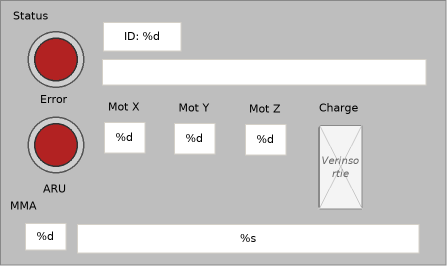
VISUALIZATION Visu2_Status  // 447x266
    Rectangle (-2,-2 447x266)
    Image (318,126 43x83), invisible if: fbAct1.xInInPos=0, image: Verinrentree
    Rectangle (320,150 37x38), "Going out", invisible if: fbAct1.xGoingOutNow=0
    Lamp1 (22,112 68x66), variable: fbBtn.xAru=0, style: Lamp-Lamp1-Red
    Lamp1 (23,25 66x69), variable: stParam.stStatus.xErreur, style: Lamp-Lamp1-Red
    Textfield (102,59 324x26), text variable: stParam.stStatus.sMessage, text list: 'ErrorList', text index: stParam.stStatus.iId
    Textfield (103,22 78x29), "ID: %d", text variable: stParam.stStatus.iId
    Label (299,93 80x30), "Charge"
    Image (319,125 43x84), invisible if: fbAct1.xInOutPos=0, image: Verinsortie
    Textfield (245,124 41x31), "%d", text variable: fbMotorZ.fbAxisRef.NcToPlc.ActPos
    Label (225,94 80x30), "Mot Z"
    Label (154,93 80x30), "Mot Y"
    Textfield (174,123 41x31), "%d", text variable: fbMotorY.fbAxisRef.NcToPlc.ActPos
    Label (84,92 80x30), "Mot X"
    Textfield (104,122 41x31), "%d", text variable: fbMotorX.fbAxisRef.NcToPlc.ActPos
    Label (10,1 176x30), "Status"
    Label (26,85 55x29), "Error"
    Label (11,175 87x28), "ARU"
    Label (7,191 80x30), "MMA"
    Textfield (77,224 342x29), "%s", text variable: fbMMA.fbEtape.sMess
    Textfield (25,223 41x27), "%d", text variable: fbMMA.iEtape
END_VISUALIZATION

(* stored: Version 1.1.0.1, ProductVersion 3.1.4020.12
   Visu Visu2_Status: Id {00e42565-6edb-4ff6-a05e-94125dfe942e} *)
